{attribute 'qualified_only'}
{attribute 'strict'}
TYPE StatusStep :
(
	Inactive,
	Active,
	Faulted,
	TimedOut,
	Complete
);
END_TYPE

(* stored: Version 1.1.0.1, ProductVersion 3.1.4022.11
   DUT StatusStep: Id {9dce691a-8e78-4e62-922f-74f081232cbf} *)
